PROGRAM PRG_PMPS
VAR
	 fbArbiterIO : FB_SubSysToArbiter_IO;

	ff2_ff1_link: FB_FastFault := (i_xAutoReset := TRUE, i_DevName := 'FF2 to FF1 Link', i_Desc := 'This is virtual FF2 fault, Please check the faulting device below', i_TypeCode := 16#9999);

END_VAR

(*Fast Fault instantiation*)
GVL_PMPS.g_FastFaultOutput1.bAutoReset :=TRUE;
GVL_PMPS.g_FastFaultOutput2.bAutoReset :=TRUE;
GVL_PMPS.g_FastFaultOutput1.Execute(i_xVeto := (PMPS_GVL.stCurrentBeamParameters.aVetoDevices[PMPS.K_Stopper.MR1K1_OUT] 
                                      AND NOT PMPS_GVL.stCurrentBeamParameters.aVetoDevices[PMPS.K_Stopper.MR1K1_IN])
                                       OR PMPS_GVL.stCurrentBeamParameters.aVetoDevices[PMPS.K_Stopper.ST1K2]);
GVL_PMPS.g_FastFaultOutput2.Execute(i_xVeto := (PMPS_GVL.stCurrentBeamParameters.aVetoDevices[PMPS.K_Stopper.MR1K1_OUT] 
                                      AND NOT PMPS_GVL.stCurrentBeamParameters.aVetoDevices[PMPS.K_Stopper.MR1K1_IN])
                                       OR PMPS_GVL.stCurrentBeamParameters.aVetoDevices[PMPS.K_Stopper.ST1K2]);
(* Arbiter Instantiation*)
fbArbiterIO(Arbiter := GVL_PMPS.fbArbiter1, fbFFHWO := GVL_PMPS.g_FastFaultOutput1, i_bVeto := (PMPS_GVL.stCurrentBeamParameters.aVetoDevices[PMPS.K_Stopper.MR1K1_OUT] 
                                      AND NOT PMPS_GVL.stCurrentBeamParameters.aVetoDevices[PMPS.K_Stopper.MR1K1_IN])
                                       OR PMPS_GVL.stCurrentBeamParameters.aVetoDevices[PMPS.K_Stopper.ST1K2]);
//routed to the arbiter							   
ff2_ff1_link(
	io_fbFFHWO := GVL_PMPS.g_FastFaultOutput2,
    i_xOK := GVL_PMPS.g_FastFaultOutput1.q_xFastFaultOut);

END_PROGRAM

(* stored: Version 1.1.0.1, ProductVersion 3.1.4022.18
   POU PRG_PMPS: Id {c0394586-ec07-4cb6-8556-b8d523a91d95}, SpecialFunc None *)
